// TIA Portal V15.1 export
// export: Created 2024-05-17T05:38:24.4171935Z, ExportSetting WithDefaults, DisplayName Totally Integrated Automation Portal, DisplayVersion V15.1 Update 5, DisplayName TIA Portal Openness, DisplayVersion V15.1 Update 5, DisplayName SINAMICS Startdrive Advanced, DisplayVersion V15.1, DisplayName G130, G150, S120, S150, SINAMICS MV, S210, DisplayVersion V15.1, DisplayName G110M, G120, G120C, G120D, G120P, DisplayVersion V15.1, DisplayName STEP 7 Professional, DisplayVersion V15.1 Update 5, DisplayName STEP 7 Safety, DisplayVersion V15.1, DisplayName WinCC Professional, DisplayVersion V15.1 Update 5, DisplayName SIMATIC Visualization Architect, DisplayVersion V15.1
FUNCTION "F209230ZS01Output" : Void   // FC7032, F_FBD
TITLE = Safety Inputs ZMProc / Safety Outputs 209230ZS01
{ S7_Optimized_Access := 'TRUE' }
VERSION : 0.1
// stored: AutoNumber false, IsIECCheckEnabled false, UDAEnableTagReadback false
BEGIN

REGION Network 1: **** 8 - Outputs **** 209230CA21M4-UE150 STO
   // SEW Drive STO
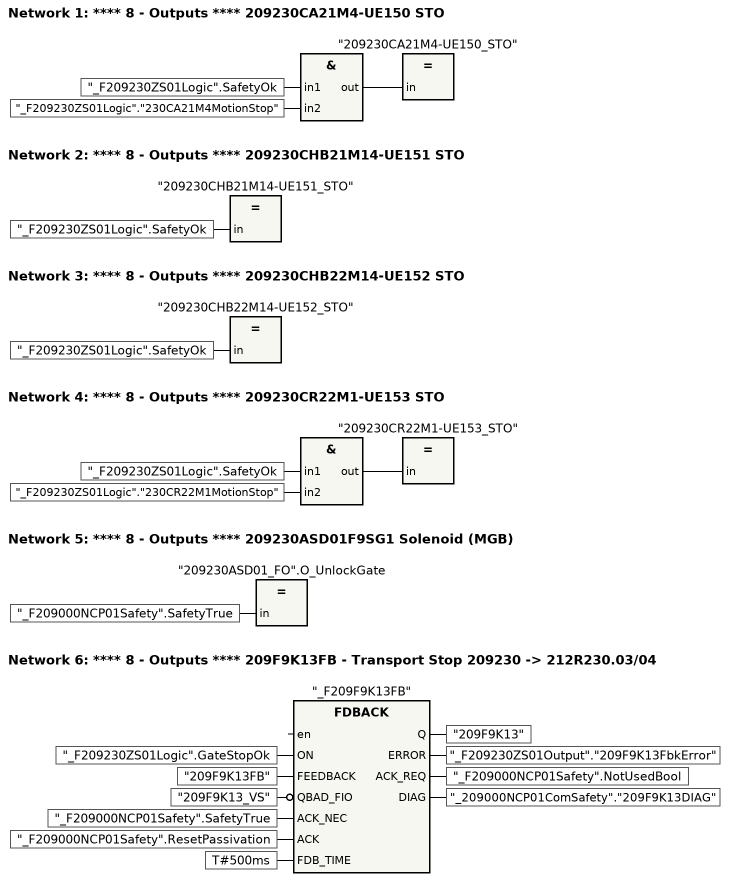
   "209230CA21M4-UE150_STO" := "_F209230ZS01Logic".SafetyOk AND "_F209230ZS01Logic"."230CA21M4MotionStop";
END_REGION

REGION Network 2: **** 8 - Outputs **** 209230CHB21M14-UE151 STO
   // SEW Drive STO
   "209230CHB21M14-UE151_STO" := "_F209230ZS01Logic".SafetyOk;
END_REGION

REGION Network 3: **** 8 - Outputs **** 209230CHB22M14-UE152 STO
   // SEW Drive STO
   "209230CHB22M14-UE152_STO" := "_F209230ZS01Logic".SafetyOk;
END_REGION

REGION Network 4: **** 8 - Outputs **** 209230CR22M1-UE153 STO
   // SEW Drive STO
   "209230CR22M1-UE153_STO" := "_F209230ZS01Logic".SafetyOk AND "_F209230ZS01Logic"."230CR22M1MotionStop";
END_REGION

REGION Network 5: **** 8 - Outputs **** 209230ASD01F9SG1 Solenoid (MGB)
   // Safety Door Solenoid
   "209230ASD01_FO".O_UnlockGate := "_F209000NCP01Safety".SafetyTrue;
END_REGION

REGION Network 6: **** 8 - Outputs **** 209F9K13FB - Transport Stop 209230 -> 212R230.03/04
   // Transport Stop 209230 -> 212R230.03/04
   "_F209F9K13FB"(ON := "_F209230ZS01Logic".GateStopOk,   // FDBACK
                  FEEDBACK := "209F9K13FB",
                  QBAD_FIO := NOT "209F9K13_VS",
                  ACK_NEC := "_F209000NCP01Safety".SafetyTrue,
                  ACK := "_F209000NCP01Safety".ResetPassivation,
                  FDB_TIME := T#500ms,
                  Q => "209F9K13",
                  ERROR => "_F209230ZS01Output"."209F9K13FbkError",
                  ACK_REQ => "_F209000NCP01Safety".NotUsedBool,
                  DIAG => "_209000NCP01ComSafety"."209F9K13DIAG");
END_REGION
END_FUNCTION
